{attribute 'GeneratedUsingTerminal: EL6201-0000-0017'}
{attribute addProperty BoxType "EL6201-0000-0017"}
{attribute addProperty Id "Slave_7A_DI0BOOL1Slave_7A_DI1BOOL1Slave_7A_DI2BOOL1Slave_7A_DI3BOOL1Slave_7B_DI0BOOL1Slave_7B_DI1BOOL1Slave_7B_DI2BOOL1Slave_7B_DI3BOOL1"}
{attribute addProperty CRC "4130235232"}
{attribute addProperty Size "8"}
TYPE Slave_7_Inputs_F62E6360 :
STRUCT
	{attribute addProperty Name "Slave_7A_DI0"}
	Slave_7A_DI0 : BOOL;
	{attribute addProperty Name "Slave_7A_DI1"}
	Slave_7A_DI1 : BOOL;
	{attribute addProperty Name "Slave_7A_DI2"}
	Slave_7A_DI2 : BOOL;
	{attribute addProperty Name "Slave_7A_DI3"}
	Slave_7A_DI3 : BOOL;
	{attribute addProperty Name "Slave_7B_DI0"}
	Slave_7B_DI0 : BOOL;
	{attribute addProperty Name "Slave_7B_DI1"}
	Slave_7B_DI1 : BOOL;
	{attribute addProperty Name "Slave_7B_DI2"}
	Slave_7B_DI2 : BOOL;
	{attribute addProperty Name "Slave_7B_DI3"}
	Slave_7B_DI3 : BOOL;
END_STRUCT
END_TYPE

(* stored: Version 1.2.0.0, ProductVersion 3.1.4024.9
   DUT Slave_7_Inputs_F62E6360: Id {4ea4d987-2a36-41e2-885a-e11ab6f3101b} *)
